// Drive share Data for sync operation with dependent FBs
INTERFACE I_MotionDriveShareData

PROPERTY DriveEnable : BOOL
SET
END_SET
END_PROPERTY

PROPERTY ExecHome : BOOL
SET
END_SET
END_PROPERTY

PROPERTY ExecMove : BOOL
SET
END_SET
END_PROPERTY

PROPERTY GlobalReset : BOOL
SET
END_SET
END_PROPERTY

PROPERTY NewMoveReq : BOOL
SET
END_SET
END_PROPERTY

PROPERTY RestoreDone : BOOL
GET
END_GET
END_PROPERTY

PROPERTY SavedPosition : LREAL
GET
END_GET
END_PROPERTY

PROPERTY ServoMode : BOOL
SET
END_SET
END_PROPERTY

END_INTERFACE

(* stored: Version 1.1.0.1
   Itf I_MotionDriveShareData: Id {9543722d-3dbe-4c87-81ba-7da492b88902}
   Property DriveEnable: Id {826cf95b-d692-439f-98da-b92ffc221680}
   Set Set: Id {640b0499-6307-45e9-81dc-5959999d6c90}
   Property ExecHome: Id {908d2746-3d7e-4ea3-b913-8e6be2904464}
   Set Set: Id {1625bc31-1b5b-40e7-9a98-7961350aee4e}
   Property ExecMove: Id {91487e24-bb27-4248-b9cb-9055edd0e028}
   Set Set: Id {5ac5283c-c89e-401a-a084-7e84ab3967ca}
   Property GlobalReset: Id {28b10428-fdb5-4e5c-8261-86290842e88e}
   Set Set: Id {dfb7a8a2-9e94-4bfc-91bd-25044dac290a}
   Property NewMoveReq: Id {2a71e750-3fad-4db0-87d3-c4b98647d7fb}
   Set Set: Id {09c8c3dd-11ef-4ead-a52e-664001a563d6}
   Property RestoreDone: Id {96c9cb56-d5db-4a71-b88e-6f41fa10fa38}
   Get Get: Id {1965c5bc-4b79-47e3-8434-562f062a9501}
   Property SavedPosition: Id {779333e4-9ab7-4cd6-a267-fa2dae801e08}
   Get Get: Id {20eff14e-209d-4a1c-b8f5-f4ae3261783e}
   Property ServoMode: Id {50a918a3-b327-4921-a8e8-6398cf7d9306}
   Set Set: Id {dea97cd8-a66f-498c-9d74-0f702b621652} *)
